INTERFACE I_DatatypePack

METHOD RegisterWithDatatypes
VAR_INPUT
	Datatypes : I_Datatypes;
END_VAR
END_METHOD

END_INTERFACE

(* stored: Version 1.1.0.1, ProductVersion 3.1.4024.12
   Itf I_DatatypePack: Id {dd3f9974-a398-0830-058a-1218022de8e2}
   Method RegisterWithDatatypes: Id {94fa4154-2078-02cb-1855-2082629990ac} *)
